FUNCTION_BLOCK Teste (* Basic FB with empty ECC *)
  (* Standard: 61499-2 *)
  (* Version 1.0, 2024-12-17, Bruno *)
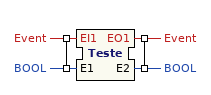
  EVENT_INPUT
    EI1 WITH E1;
  END_EVENT
  EVENT_OUTPUT
    EO1 WITH E2;
  END_EVENT
  VAR_INPUT
    E1 : BOOL;
  END_VAR
  VAR_OUTPUT
    E2 : BOOL;
  END_VAR
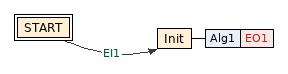
  EC_STATES
    START; (* Initial State *)
    Init : Alg1 -> EO1;
  END_STATES
  EC_TRANSITIONS
    START TO Init := EI1;
  END_TRANSITIONS
  ALGORITHM Alg1 IN ST:
E2 := NOT E2;
  END_ALGORITHM
END_FUNCTION_BLOCK
